// TIA Portal V18 export
VAR_GLOBAL   // PLC tag table "05_RD-1"
   "iRD-1" AT %I1.2 : Bool;
   "oRD-1" AT %Q0.4 : Bool;
END_VAR
